# EPICS substitutions: db/Beckhoff_5XXX/ecmcEL5101_32bit.substitutions
file "ecmcEL5101-chX.template"
{
    pattern {CH_ID}
            {01   }
}

# Period and frequency measurement
file "ecmcEL5101-chX_32bit_extras.template"
{
  pattern {CH_ID}
          {01   }
}
